# EPICS substitutions: ek9000App/Db/EL4031.substitutions
file EL4031.template
{       pattern
        {
                TERMINAL,

        }
        {
        }
}
